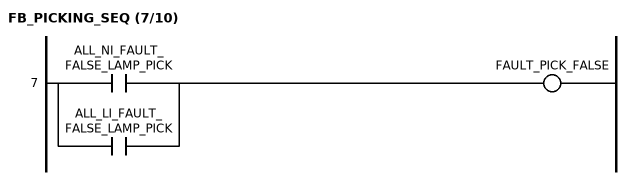
(* [picture p48: FB_PICKING_SEQ, rungs 7-7] *)
(* Rung 7 *)
FAULT_PICK_FALSE := ALL_NI_FAULT_FALSE_LAMP_PICK OR ALL_LI_FAULT_FALSE_LAMP_PICK;

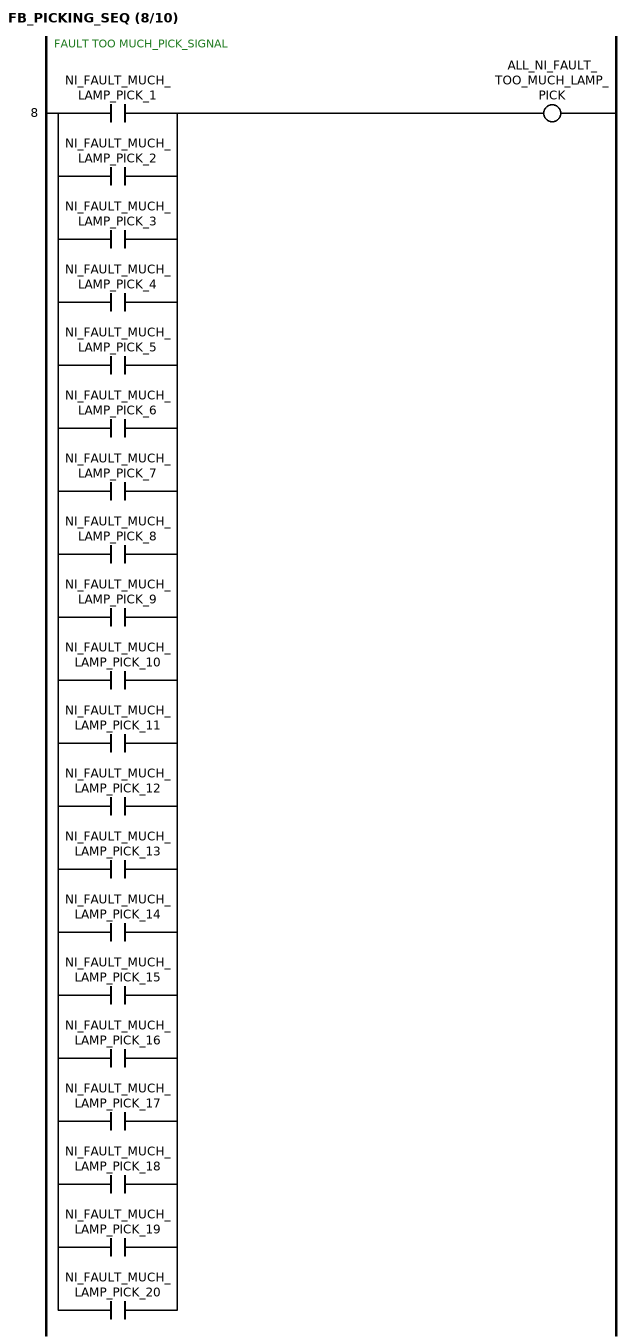
(* Rung 8: FAULT TOO MUCH_PICK_SIGNAL *)
ALL_NI_FAULT_TOO_MUCH_LAMP_PICK := NI_FAULT_MUCH_LAMP_PICK_1 OR NI_FAULT_MUCH_LAMP_PICK_2 OR NI_FAULT_MUCH_LAMP_PICK_3 OR NI_FAULT_MUCH_LAMP_PICK_4 OR NI_FAULT_MUCH_LAMP_PICK_5 OR NI_FAULT_MUCH_LAMP_PICK_6 OR NI_FAULT_MUCH_LAMP_PICK_7 OR NI_FAULT_MUCH_LAMP_PICK_8 OR NI_FAULT_MUCH_LAMP_PICK_9 OR NI_FAULT_MUCH_LAMP_PICK_10 OR NI_FAULT_MUCH_LAMP_PICK_11 OR NI_FAULT_MUCH_LAMP_PICK_12 OR NI_FAULT_MUCH_LAMP_PICK_13 OR NI_FAULT_MUCH_LAMP_PICK_14 OR NI_FAULT_MUCH_LAMP_PICK_15 OR NI_FAULT_MUCH_LAMP_PICK_16 OR NI_FAULT_MUCH_LAMP_PICK_17 OR NI_FAULT_MUCH_LAMP_PICK_18 OR NI_FAULT_MUCH_LAMP_PICK_19 OR NI_FAULT_MUCH_LAMP_PICK_20;

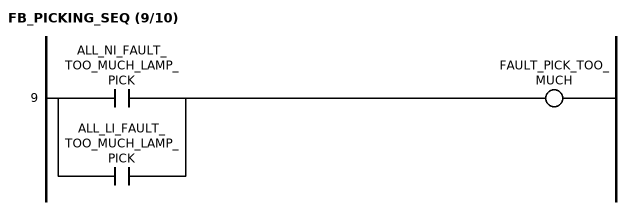
(* Rung 9 *)
FAULT_PICK_TOO_MUCH := ALL_NI_FAULT_TOO_MUCH_LAMP_PICK OR ALL_LI_FAULT_TOO_MUCH_LAMP_PICK;

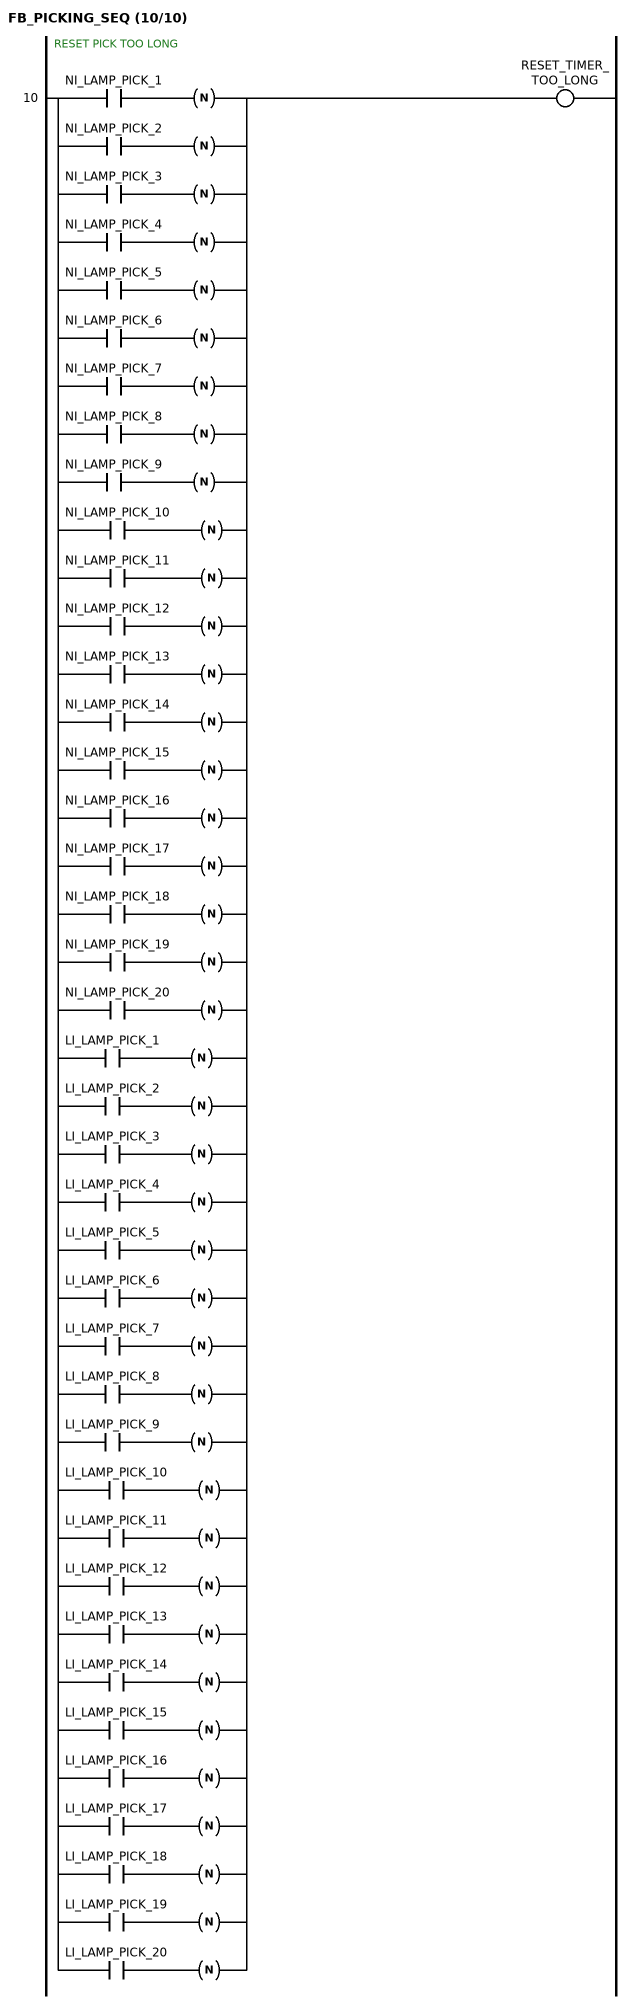
(* Rung 10: RESET PICK TOO LONG *)
_e92(CLK := NI_LAMP_PICK_1);
_e93(CLK := NI_LAMP_PICK_2);
_e94(CLK := NI_LAMP_PICK_3);
_e95(CLK := NI_LAMP_PICK_4);
_e96(CLK := NI_LAMP_PICK_5);
_e97(CLK := NI_LAMP_PICK_6);
_e98(CLK := NI_LAMP_PICK_7);
_e99(CLK := NI_LAMP_PICK_8);
_e100(CLK := NI_LAMP_PICK_9);
_e101(CLK := NI_LAMP_PICK_10);
_e102(CLK := NI_LAMP_PICK_11);
_e103(CLK := NI_LAMP_PICK_12);
_e104(CLK := NI_LAMP_PICK_13);
_e105(CLK := NI_LAMP_PICK_14);
_e106(CLK := NI_LAMP_PICK_15);
_e107(CLK := NI_LAMP_PICK_16);
_e108(CLK := NI_LAMP_PICK_17);
_e109(CLK := NI_LAMP_PICK_18);
_e110(CLK := NI_LAMP_PICK_19);
_e111(CLK := NI_LAMP_PICK_20);
_e112(CLK := LI_LAMP_PICK_1);
_e113(CLK := LI_LAMP_PICK_2);
_e114(CLK := LI_LAMP_PICK_3);
_e115(CLK := LI_LAMP_PICK_4);
_e116(CLK := LI_LAMP_PICK_5);
_e117(CLK := LI_LAMP_PICK_6);
_e118(CLK := LI_LAMP_PICK_7);
_e119(CLK := LI_LAMP_PICK_8);
_e120(CLK := LI_LAMP_PICK_9);
_e121(CLK := LI_LAMP_PICK_10);
_e122(CLK := LI_LAMP_PICK_11);
_e123(CLK := LI_LAMP_PICK_12);
_e124(CLK := LI_LAMP_PICK_13);
_e125(CLK := LI_LAMP_PICK_14);
_e126(CLK := LI_LAMP_PICK_15);
_e127(CLK := LI_LAMP_PICK_16);
_e128(CLK := LI_LAMP_PICK_17);
_e129(CLK := LI_LAMP_PICK_18);
_e130(CLK := LI_LAMP_PICK_19);
_e131(CLK := LI_LAMP_PICK_20);
RESET_TIMER_TOO_LONG := _e92.Q OR _e93.Q OR _e94.Q OR _e95.Q OR _e96.Q OR _e97.Q OR _e98.Q OR _e99.Q OR _e100.Q OR _e101.Q OR _e102.Q OR _e103.Q OR _e104.Q OR _e105.Q OR _e106.Q OR _e107.Q OR _e108.Q OR _e109.Q OR _e110.Q OR _e111.Q OR _e112.Q OR _e113.Q OR _e114.Q OR _e115.Q OR _e116.Q OR _e117.Q OR _e118.Q OR _e119.Q OR _e120.Q OR _e121.Q OR _e122.Q OR _e123.Q OR _e124.Q OR _e125.Q OR _e126.Q OR _e127.Q OR _e128.Q OR _e129.Q OR _e130.Q OR _e131.Q;
END_FUNCTION_BLOCK